ABB RobotStudio station: Solution2_20190820-231001.rsstn

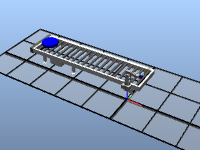
Station Solution2 (saved by RobotStudio 7.0.8504.151)
Controller Vinnie, task T_ROB1: task frame (RAPID world) sits at (0, 0, 400) mm in the station
Controller Vinnie
  mechanical unit ROB_1: IRB120_3_58__01, 6 joints, base frame (0, 0, 0) mm
Layout (positions relative to the parent item):
  - IRB120_3_58__01 [mechanism, from Robots\IRB120_3_58_G_01.rslib] at (0, 0, 400) mm; joint values [0, 0, 0, 0, 0, 0] (rad or m)
  - Conveyor1 [smart component]
      signals: DI NewBox, DO BoxAtPos
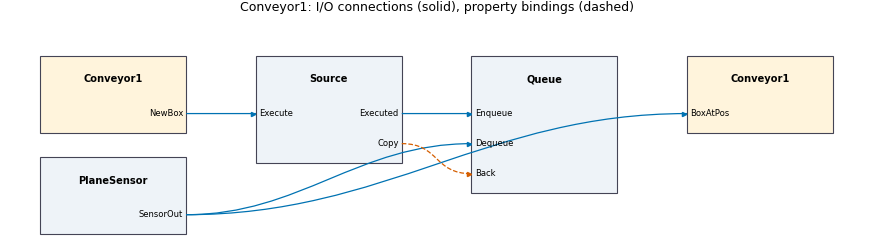
      connections:
        Conveyor1.NewBox -> Source.Execute
        Source.Executed -> Queue.Enqueue
        PlaneSensor.SensorOut -> Queue.Dequeue
        PlaneSensor.SensorOut -> Conveyor1.BoxAtPos
        Source.Copy => Queue.Back
    - 950_4000_h2 [part, from Equipment\Conveyor 950 4000 h2.rslib] at (-3846.63, 300, 0) mm
    - Source [smart component, from Components\Source.rslib]
        properties: Source=Cylinder_300_100; Copy=(none); Parent=(none); Position=[0 0 0]; Orientation=[0 0 0]; Transient=false; PhysicsBehavior=0
    - Queue [smart component, from Components\Queue.rslib]
        properties: Back=(none); Front=(none); Queue={9d28df3f-1262-4b7a-ac04-edcd9d5f27b5};{863827ec-ac74-4948-8b9a-7544d75eb816};{d5b0fd52-96a2-4c78-9daf-449b82394716};{cae2c484-551c-4e63-899e-3f16cc655c36};{2cd56b75-4092-4768-a475-00f35c4dae8b};{e0dd32b4-5c51-4f0d-a48d-accb6fe5d5c2}; NumberOfObjects=1
    - LinearMover [smart component, from Components\LinearMover.rslib]
        properties: Object=Queue; Direction=[1 0 0]; Speed=0.5; Reference=Global; ReferenceObject=(none)
    - PlaneSensor [smart component, from Components\PlaneSensor.rslib]
        properties: Origin=[0.162459 1.21 0.435]; Axis1=[0 -0.91 0]; Axis2=[0 0 0.2]; SensedPart=(none)
      - _sensorPart_ [part]
  - Cylinder_300_100 [part, from Training Objects\my_cl.rslib] at (-3535.01, 824.34, 414.67) mm
